Fanuc TP program (LS listing): DOOR_OP_COND.LS

/PROG  DOOR_OP_COND	  Cond
/ATTR
OWNER		= MNEDITOR;
COMMENT		= "monitor";
PROG_SIZE	= 164;
CREATE		= DATE 25-07-16  TIME 20:52:56;
MODIFIED	= DATE 25-07-16  TIME 20:55:12;
FILE_NAME	= ;
VERSION		= 0;
LINE_COUNT	= 1;
MEMORY_SIZE	= 540;
PROTECT		= READ_WRITE;
TCD:  STACK_SIZE	= 0,
      TASK_PRIORITY	= 50,
      TIME_SLICE	= 0,
      BUSY_LAMP_OFF	= 0,
      ABORT_REQUEST	= 0,
      PAUSE_REQUEST	= 0;
DEFAULT_GROUP	= *,*,*,*,*;
CONTROL_CODE	= 00000000 00000000;
/MN
   1:  WHEN DI[5:OFF:door opened]=OFF,CALL DOOR_NOT_OP ;
/POS
/END
